# EPICS substitutions: rsaApp/Db/user.substitutions
# Example substitutions file

file "db/dbExample1.db" {
    { user = "joao" }
}

file db/dbExample2.db {
    pattern { user, no, scan }
        { "joao", 1, "1 second" }
        { "joao", 2, "2 second" }
        { "joao", 3, "5 second" }
}
